TYPE ST_Ledstrip_get :
STRUCT
	b_error		: BOOL;
	BeckhoffLed	: BOOL;
END_STRUCT
END_TYPE

(* stored: Version 1.1.0.1, ProductVersion 3.1.4026.18
   DUT ST_Ledstrip_get: Id {25061d8f-abe5-4cf6-84a4-661bb1b441f0} *)
